FUNCTION_BLOCK EL3255
VAR
	_io : EL3xx5_Data;
	{attribute addProperty Name "WcState"}
	_wcState : WcStateInputToggle;
	{attribute addProperty Name "Info data"}
	_infoData : InfoDataAds;
END_VAR

PROPERTY IO : REFERENCE TO EL3xx5_Data
GET
IO REF= _io;
END_GET
END_PROPERTY

PROPERTY WcState : REFERENCE TO WcStateInputToggle
GET
WcState REF= _wcState;
END_GET
END_PROPERTY

END_FUNCTION_BLOCK

(* stored: Version 1.1.0.1, ProductVersion 3.1.4024.9
   POU EL3255: Id {e486d387-27c8-074e-0b16-eeb703368e81}, SpecialFunc None
   Property IO: Id {8f347151-3c5f-0309-32c0-34275d4a7d66}
   Get Get: Id {5ace10fd-e2e3-0c67-0cb6-8b2fb7788fb3}
   Property WcState: Id {74bc412c-d49e-08f4-22c4-97231d8c9f94}
   Get Get: Id {a09dc6be-5a77-0540-27a7-2b1f7253dab2} *)
